FUNCTION_BLOCK ABSTRACT Mc3MotionTask IMPLEMENTS I_Mc3MotionTask
VAR
	_Name : T_MaxString;
	_Axis : I_Mc3Axis;
END_VAR

PROPERTY Axis : I_Mc3Axis
GET
Axis := _Axis;
END_GET
SET
_Axis := Axis;
END_SET
END_PROPERTY

{attribute 'monitoring' := 'call'}
PROPERTY ABSTRACT Busy : BOOL
GET
END_GET
END_PROPERTY

METHOD ABSTRACT CyclicLogic
END_METHOD

{attribute 'monitoring' := 'call'}
PROPERTY ABSTRACT Error : BOOL
GET
END_GET
END_PROPERTY

{attribute 'monitoring' := 'call'}
PROPERTY ABSTRACT ErrorId : UDINT
GET
END_GET
END_PROPERTY

METHOD ABSTRACT Execute : BOOL;
END_METHOD

{attribute 'monitoring' := 'call'}
PROPERTY Name : T_MaxString
GET
Name := _Name;
END_GET
SET
_Name := Name;
END_SET
END_PROPERTY

END_FUNCTION_BLOCK

(* stored: Version 1.1.0.1, ProductVersion 3.1.4026.20
   POU Mc3MotionTask: Id {1c0d5331-b86c-495b-a2de-30799356861e}, SpecialFunc None
   Property Axis: Id {a5830217-434e-47ff-b128-792666fbdec4}
   Get Get: Id {1082a1b5-c826-4720-a9b3-1fba2f1e61a4}
   Set Set: Id {31b86d11-1ec1-4740-bb2a-8f2a481a6557}
   Property Busy: Id {93da074f-3958-496e-8e5d-1260a89e6e0a}
   Get Get: Id {cb637ede-0538-4d50-82cb-90d0d6464416}
   Method CyclicLogic: Id {fa4acd00-f801-4908-98a7-381e63544e87}
   Property Error: Id {67194bfb-7674-45f0-8ce0-ebab9a751cb2}
   Get Get: Id {e8d97a86-f459-4412-9b34-37246e6d8e02}
   Property ErrorId: Id {6766c30e-3515-43ed-982a-82e17815a2ed}
   Get Get: Id {392451d8-dba6-4e41-898a-95d8b5cb3a16}
   Method Execute: Id {cc134bcd-5bde-4d4f-9c29-080882c25ba4}
   Property Name: Id {aea1bd0f-4d2f-433c-8a9e-06adb5ea7537}
   Get Get: Id {7595e056-5d25-4592-a4cf-1ba58b00eaea}
   Set Set: Id {05a0394f-5541-4cb0-8758-d6fd2d7cf403} *)
